// This Function is used to avoid division by 0.
// If you integrate these functions in the PLC project, they are called before each division that occurs in the code.
// Implicitly generated code : DO NOT EDIT
FUNCTION CheckDivLInt : LINT
VAR_INPUT
	divisor:LINT;
END_VAR

// Implicitly generated code : Only an Implementation suggestion
{noflow}
IF divisor = 0 THEN
	CheckDivLInt:=1;
	GVL_TwinCatChecks.CheckDiv_LINT_DivBy0 := GVL_TwinCatChecks.CheckDiv_LINT_DivBy0 + 1;
ELSE
	CheckDivLInt:=divisor;
END_IF;
{flow}

END_FUNCTION

(* stored: Version 1.1.0.1
   POU CheckDivLInt: Id {462be0e7-2ad6-4726-8275-21e7b020987c}, SpecialFunc CheckDivInt64 *)
